TYPE DUT_MotorFeedbackSnapshot : STRUCT
    encoder_position_raw       : DINT;
    encoder_velocity_raw       : DINT;
    copley_statusword          : WORD;
    copley_actual_current_count: INT;
    output_torque_count        : INT;
    fault_id                   : UDINT;
END_STRUCT
END_TYPE

(* stored: Version 1.1.0.1, ProductVersion 3.1.4024.12
   DUT DUT_MotorFeedbackSnapshot: Id {9f95b821-e6f9-4e51-98dd-900047a01002} *)
